// TIA Portal V19 export
// export: Created 2024-12-12T07:14:07.305667Z, ExportSetting WithDefaults, DisplayName Totally Integrated Automation Portal, DisplayVersion V19 Update 1, DisplayName TIA Portal Openness, DisplayVersion V19 Update 1, DisplayName TIA Portal Version Control Interface, DisplayVersion V19, DisplayName SINAMICS Startdrive Advanced, DisplayVersion V19, DisplayName SINAMICS DCC, DisplayVersion V19, DisplayName SINAMICS Startdrive G130, G150, S120, S150, SINAMICS MV, G220, S200, S210, DisplayVersion V19, DisplayName SINAMICS Startdrive G110M, G120, G120C, G120D, G120P, G115D, DisplayVersion V19, DisplayName STEP 7 Professional, DisplayVersion V19 Update 1, DisplayName STEP 7 Safety, DisplayVersion V19 Update 1, DisplayName WinCC Advanced, DisplayVersion V19 Update 1, DisplayName WinCC Advanced / Unified PC, DisplayVersion V19 Update 1
DATA_BLOCK "CW1"   // DB218
{ S7_Optimized_Access := 'TRUE' }
VERSION : 0.1
// stored: AutoNumber true, DBAccessibleFromOPCUA true, DBAccessibleFromWebserver true, InstanceOfName EM_CWM, InstanceOfType UDT, IsOnlyStoredInLoadMemory false, IsWriteProtectedInAS false
"EM_CWM"
   // VAR RETAIN
   //    Std : "EM_Std";
   //    Param : "EM_CWM_Param";
   //    LastHmiDataParam : "EM_CWM_Param";
   //    Alm : "EM_CWM_Alm";
   //    AlmWinCC : "EM_CWM_AlmWinCC";
   //    Sign : "EM_Sign";
   //    SignWinCC : "EM_Sign_WinCC";
   //    Input : "EM_CWM_Input";
   //    Output : "EM_CWM_Output";
   //    ExchangeFromChain : "EM_CWM_Exchange_FromChain";
   //    ExchangeToChain : "EM_CWM_Exchange_ToChain";
   //    Scale : "Scale_Wipotec";
   // END_VAR
BEGIN
   Std.Cfg_ModuleSync := TRUE;
   Std.Cfg_0_BelongShort_1_BelongLong := TRUE;
   Std.Cfg_ExternalCPU := FALSE;
   Std.Cfg_0_JogWord_1_JogBit := TRUE;
   Std._0_PriorityAlm_1_FirstAlm := FALSE;
   Std.AbortAlmOk := TRUE;
   Std.ServicesAbortAlmOk := TRUE;
   Std.SignOK := TRUE;
   Std.AlmReset := FALSE;
   Std.SignReset := FALSE;
   Std.NewAlm := FALSE;
   Std.NewSign := FALSE;
   Std.RstNewAlm := FALSE;
   Std.RstNewSign := FALSE;
   Std.AllowCopyByCategory := TRUE;
   Std.ForceCopyAll := FALSE;
   Std.InitCategories := FALSE;
   Std.InitCauses := FALSE;
   Std.Diag_AlmFound := FALSE;
   Std.Diag_SignFound := FALSE;
   Std.ScOk := TRUE;
   Std.OkToStop := TRUE;
   Std.PwrDrv := TRUE;
   Std.DriveRunCmd := FALSE;
   Std.ManAct := FALSE;
   Std.MachineSelected := TRUE;
   Std.MachineExtracted := FALSE;
   Std.LocalAbortReq := FALSE;
   Std.CondOkToEnaStaReq := FALSE;
   Std.EnaReq := FALSE;
   Std.EnaStaReq := FALSE;
   Std.StaReq := FALSE;
   Std.ReqStart := FALSE;
   Std.ReqStop := FALSE;
   Std.ReqAbort := TRUE;
   Std.ReqExecute := FALSE;
   Std.ReqReset := FALSE;
   Std.ReqSuspend := FALSE;
   Std.ReqUnSuspend := FALSE;
   Std.StrobeDeviceDiag := TRUE;
   Std.StrobeInverterDiag := FALSE;
   Std.DeviceDiagnosticDone := FALSE;
   Std.InverterDiagnosticDone := FALSE;
   Std.RecipeOnlineLoadDone := FALSE;
   Std.RecipeOnlineSaveDone := FALSE;
   Std.RecipeOfflineLoadDone := FALSE;
   Std.RecipeOfflineSaveDone := FALSE;
   Std.LastHmiDataLoadDone := FALSE;
   Std.LastHmiDataSaveDone := FALSE;
   Std.SummAlmTimeoutStart := FALSE;
   Std.SirenEna := FALSE;
   Std.VisEnButtons := TRUE;
   Std.VisManButtons := FALSE;
   Std.VisHomeButtons := FALSE;
   Std.VisEnButtonsRunning := TRUE;
   Std.Ena_Suspended := TRUE;
   Std.BluStkLgh_Steady_Cond := FALSE;
   Std.BluStkLgh_Frequency1_Cond := FALSE;
   Std.Siren_Frequency4_Cond := FALSE;
   Std.Cfg_ModuleNumber := 5;
   Std.Cfg_DeviceDiagCounter_Preset := 1;
   Std.Cfg_InverterDiagCounter_Preset := 0;
   Std.Cfg_Num_AlmDint := 8;
   Std.Cfg_Num_SignDint := 3;
   Std.Cfg_StaPbt := 65535;
   Std.Cfg_StoPbt := 65535;
   Std.Cfg_RstPbt := -1;
   Std.Cfg_EnaPbt := 65535;
   Std.Cfg_Siren := 1;
   Std.Cfg_Stack := 1;
   Std.Cfg_DisableStates[0..31] := 0;
   Std.Cfg_ModeTransitions[0..31] := 0;
   Std.Cfg_ModeNames[0..31] := '';
   Std.ModeCurrentName := 'Production';
   Std.StateCurrentName := 'Aborted';
   Std.DeviceDiagCounter := 1;
   Std.InverterDiagCounter := 0;
   Std.MaintenanceActivated."0" := FALSE;
   Std.MaintenanceActivated."1" := FALSE;
   Std.MaintenanceActivated."2" := FALSE;
   Std.MaintenanceActivated."3" := FALSE;
   Std.MaintenanceActivated."4" := FALSE;
   Std.MaintenanceActivated."5" := FALSE;
   Std.MaintenanceActivated."6" := FALSE;
   Std.MaintenanceActivated."7" := FALSE;
   Std.MaintenanceActivated."8" := FALSE;
   Std.MaintenanceActivated."9" := FALSE;
   Std.MaintenanceActivated."10" := FALSE;
   Std.MaintenanceActivated."11" := FALSE;
   Std.MaintenanceActivated."12" := FALSE;
   Std.MaintenanceActivated."13" := FALSE;
   Std.MaintenanceActivated."14" := FALSE;
   Std.MaintenanceActivated."15" := FALSE;
   Std.MaintenanceActivated."16" := FALSE;
   Std.MaintenanceActivated."17" := FALSE;
   Std.MaintenanceActivated."18" := FALSE;
   Std.MaintenanceActivated."19" := FALSE;
   Std.MaintenanceActivated."20" := FALSE;
   Std.MaintenanceActivated."21" := FALSE;
   Std.MaintenanceActivated."22" := FALSE;
   Std.MaintenanceActivated."23" := FALSE;
   Std.MaintenanceActivated."24" := FALSE;
   Std.MaintenanceActivated."25" := FALSE;
   Std.MaintenanceActivated."26" := FALSE;
   Std.MaintenanceActivated."27" := FALSE;
   Std.MaintenanceActivated."28" := FALSE;
   Std.MaintenanceActivated."29" := FALSE;
   Std.MaintenanceActivated."30" := FALSE;
   Std.MaintenanceActivated."31" := FALSE;
   Std.MaintenanceReq."0" := FALSE;
   Std.MaintenanceReq."1" := FALSE;
   Std.MaintenanceReq."2" := FALSE;
   Std.MaintenanceReq."3" := FALSE;
   Std.MaintenanceReq."4" := FALSE;
   Std.MaintenanceReq."5" := FALSE;
   Std.MaintenanceReq."6" := FALSE;
   Std.MaintenanceReq."7" := FALSE;
   Std.MaintenanceReq."8" := FALSE;
   Std.MaintenanceReq."9" := FALSE;
   Std.MaintenanceReq."10" := FALSE;
   Std.MaintenanceReq."11" := FALSE;
   Std.MaintenanceReq."12" := FALSE;
   Std.MaintenanceReq."13" := FALSE;
   Std.MaintenanceReq."14" := FALSE;
   Std.MaintenanceReq."15" := FALSE;
   Std.MaintenanceReq."16" := FALSE;
   Std.MaintenanceReq."17" := FALSE;
   Std.MaintenanceReq."18" := FALSE;
   Std.MaintenanceReq."19" := FALSE;
   Std.MaintenanceReq."20" := FALSE;
   Std.MaintenanceReq."21" := FALSE;
   Std.MaintenanceReq."22" := FALSE;
   Std.MaintenanceReq."23" := FALSE;
   Std.MaintenanceReq."24" := FALSE;
   Std.MaintenanceReq."25" := FALSE;
   Std.MaintenanceReq."26" := FALSE;
   Std.MaintenanceReq."27" := FALSE;
   Std.MaintenanceReq."28" := FALSE;
   Std.MaintenanceReq."29" := FALSE;
   Std.MaintenanceReq."30" := FALSE;
   Std.MaintenanceReq."31" := FALSE;
   Std.WithinScreenRange := 0;
   Std.ExchangeToGlobal.Communication.RunMode := FALSE;
   Std.ExchangeToGlobal.Communication.ConnectionFaulted := FALSE;
   Std.ExchangeToGlobal.Gen.Communication := FALSE;
   Std.ExchangeToGlobal.Gen.Selected := TRUE;
   Std.ExchangeToGlobal.Gen.Extracted := FALSE;
   Std.ExchangeToGlobal.Gen.EnaReq := FALSE;
   Std.ExchangeToGlobal.Gen.StaReq := FALSE;
   Std.ExchangeToGlobal.Gen.Started := FALSE;
   Std.ExchangeToGlobal.Gen.Unsuspended := FALSE;
   Std.ExchangeToGlobal.Gen.Ena_Suspended := TRUE;
   Std.ExchangeToGlobal.Gen.sts_Starting := FALSE;
   Std.ExchangeToGlobal.Gen.sts_Stopping := FALSE;
   Std.ExchangeToGlobal.Gen.sts_Aborting := FALSE;
   Std.ExchangeToGlobal.Gen.sts_Suspending := FALSE;
   Std.ExchangeToGlobal.Gen.sts_Unsuspending := FALSE;
   Std.ExchangeToGlobal.Gen.sts_Execute := FALSE;
   Std.ExchangeToGlobal.Gen.sts_Idle := FALSE;
   Std.ExchangeToGlobal.Gen.sts_Stopped := FALSE;
   Std.ExchangeToGlobal.Gen.sts_Aborted := TRUE;
   Std.ExchangeToGlobal.Gen.sts_Suspended := FALSE;
   Std.ExchangeToGlobal.Gen.sts_ModeManual := FALSE;
   Std.ExchangeToGlobal.Gen.sts_ModeAutomatic := TRUE;
   Std.ExchangeToGlobal.Gen.NewAlm := FALSE;
   Std.ExchangeToGlobal.Gen.NewSign := FALSE;
   Std.ExchangeToGlobal.Gen.RecipeOnlineLoadDone := FALSE;
   Std.ExchangeToGlobal.Gen.RecipeOnlineSaveDone := FALSE;
   Std.ExchangeToGlobal.Gen.RecipeOfflineLoadDone := FALSE;
   Std.ExchangeToGlobal.Gen.RecipeOfflineSaveDone := FALSE;
   Std.ExchangeToGlobal.Gen.LastHmiDataLoadDone := FALSE;
   Std.ExchangeToGlobal.Gen.LastHmiDataSaveDone := FALSE;
   Std.ExchangeToGlobal.Gen.InverterDiagnosticDone := FALSE;
   Std.ExchangeToGlobal.Gen.AxisGroupSync := TRUE;
   Std.ExchangeToGlobal.Gen.CmdMode := 1;
   Std.ExchangeToGlobal.Gen.Mode := 1;
   Std.ExchangeToGlobal.Gen.DisableEnaPbt := 0;
   Std.ExchangeToGlobal.Input.StaPbt := FALSE;
   Std.ExchangeToGlobal.Input.StoPbt := FALSE;
   Std.ExchangeToGlobal.Input.RstPbt := FALSE;
   Std.ExchangeToGlobal.Input.EnaPbt := FALSE;
   Std.ExchangeToGlobal.Input._4 := FALSE;
   Std.ExchangeToGlobal.Input._5 := FALSE;
   Std.ExchangeToGlobal.Input._6 := FALSE;
   Std.ExchangeToGlobal.Input._7 := FALSE;
   Std.ExchangeToGlobal.Input._8 := FALSE;
   Std.ExchangeToGlobal.Input._9 := FALSE;
   Std.ExchangeToGlobal.Input._10 := FALSE;
   Std.ExchangeToGlobal.Input._11 := FALSE;
   Std.ExchangeToGlobal.Input._12 := FALSE;
   Std.ExchangeToGlobal.Input._13 := FALSE;
   Std.ExchangeToGlobal.Input._14 := FALSE;
   Std.ExchangeToGlobal.Input._15 := FALSE;
   Std.ExchangeToGlobal.AlmOk.ThSwitch := TRUE;
   Std.ExchangeToGlobal.AlmOk.SafeComm := TRUE;
   Std.ExchangeToGlobal.AlmOk.SafeEmg := TRUE;
   Std.ExchangeToGlobal.AlmOk.SafeGuards := TRUE;
   Std.ExchangeToGlobal.AlmOk.GtaAirGroup := TRUE;
   Std.ExchangeToGlobal.AlmOk.Major := TRUE;
   Std.ExchangeToGlobal.AlmOk.Minor := TRUE;
   Std.ExchangeToGlobal.AlmOk.Spare07 := TRUE;
   Std.ExchangeToGlobal.AlmOk.Spare08 := TRUE;
   Std.ExchangeToGlobal.AlmOk.Spare09 := TRUE;
   Std.ExchangeToGlobal.AlmOk.Spare10 := TRUE;
   Std.ExchangeToGlobal.AlmOk.Spare11 := TRUE;
   Std.ExchangeToGlobal.AlmOk.Spare12 := TRUE;
   Std.ExchangeToGlobal.AlmOk.Spare13 := TRUE;
   Std.ExchangeToGlobal.AlmOk.Spare14 := TRUE;
   Std.ExchangeToGlobal.AlmOk.Spare15 := TRUE;
   Std.ExchangeToGlobal.AlmOk.Spare16 := TRUE;
   Std.ExchangeToGlobal.AlmOk.Spare17 := TRUE;
   Std.ExchangeToGlobal.AlmOk.Spare18 := TRUE;
   Std.ExchangeToGlobal.AlmOk.Spare19 := TRUE;
   Std.ExchangeToGlobal.AlmOk.Spare20 := TRUE;
   Std.ExchangeToGlobal.AlmOk.Spare21 := TRUE;
   Std.ExchangeToGlobal.AlmOk.Spare22 := TRUE;
   Std.ExchangeToGlobal.AlmOk.Spare23 := TRUE;
   Std.ExchangeToGlobal.AlmOk.Spare24 := TRUE;
   Std.ExchangeToGlobal.AlmOk.Spare25 := TRUE;
   Std.ExchangeToGlobal.AlmOk.Spare26 := TRUE;
   Std.ExchangeToGlobal.AlmOk.Spare27 := TRUE;
   Std.ExchangeToGlobal.AlmOk.Spare28 := TRUE;
   Std.ExchangeToGlobal.AlmOk.Spare29 := TRUE;
   Std.ExchangeToGlobal.AlmOk.Spare30 := TRUE;
   Std.ExchangeToGlobal.AlmOk.Spare31 := TRUE;
   Std.ExchangeToGlobal.AlmCauseOk.Ope := TRUE;
   Std.ExchangeToGlobal.AlmCauseOk.Ust := TRUE;
   Std.ExchangeToGlobal.AlmCauseOk.Dst := TRUE;
   Std.ExchangeToGlobal.AlmCauseOk.Ext := TRUE;
   Std.ExchangeToGlobal.AlmCauseOk.Mac := TRUE;
   Std.ExchangeToGlobal.AlmCauseOk.Spare05 := TRUE;
   Std.ExchangeToGlobal.AlmCauseOk.Spare06 := TRUE;
   Std.ExchangeToGlobal.AlmCauseOk.Spare07 := TRUE;
   Std.ExchangeToGlobal.AlmCauseOk.Spare08 := TRUE;
   Std.ExchangeToGlobal.AlmCauseOk.Spare09 := TRUE;
   Std.ExchangeToGlobal.AlmCauseOk.Spare10 := TRUE;
   Std.ExchangeToGlobal.AlmCauseOk.Spare11 := TRUE;
   Std.ExchangeToGlobal.AlmCauseOk.Spare12 := TRUE;
   Std.ExchangeToGlobal.AlmCauseOk.Spare13 := TRUE;
   Std.ExchangeToGlobal.AlmCauseOk.Spare14 := TRUE;
   Std.ExchangeToGlobal.AlmCauseOk.Spare15 := TRUE;
   Std.ExchangeToGlobal.AlmCauseOk.Spare16 := TRUE;
   Std.ExchangeToGlobal.AlmCauseOk.Spare17 := TRUE;
   Std.ExchangeToGlobal.AlmCauseOk.Spare18 := TRUE;
   Std.ExchangeToGlobal.AlmCauseOk.Spare19 := TRUE;
   Std.ExchangeToGlobal.AlmCauseOk.Spare20 := TRUE;
   Std.ExchangeToGlobal.AlmCauseOk.Spare21 := TRUE;
   Std.ExchangeToGlobal.AlmCauseOk.Spare22 := TRUE;
   Std.ExchangeToGlobal.AlmCauseOk.Spare23 := TRUE;
   Std.ExchangeToGlobal.AlmCauseOk.Spare24 := TRUE;
   Std.ExchangeToGlobal.AlmCauseOk.Spare25 := TRUE;
   Std.ExchangeToGlobal.AlmCauseOk.Spare26 := TRUE;
   Std.ExchangeToGlobal.AlmCauseOk.Spare27 := TRUE;
   Std.ExchangeToGlobal.AlmCauseOk.Spare28 := TRUE;
   Std.ExchangeToGlobal.AlmCauseOk.Spare29 := TRUE;
   Std.ExchangeToGlobal.AlmCauseOk.Spare30 := TRUE;
   Std.ExchangeToGlobal.AlmCauseOk.Spare31 := TRUE;
   Std.ExchangeToGlobal.AlmBannerFbk.FirstAlmDetection := FALSE;
   Std.ExchangeToGlobal.AlmBannerFbk.AlmPriority := 100;
   Std.ExchangeToGlobal.AlmBannerFbk.AlmCategory := -1;
   Std.ExchangeToGlobal.AlmBannerFbk.AlmCause := -1;
   Std.ExchangeToGlobal.AlmBannerFbk.AlmID := -1;
   Std.ExchangeToGlobal.AlmBannerFbk.GlobalAbsTime := 0;
   Std.ExchangeToGlobal.SignBannerFbk.SignPriority := 100;
   Std.ExchangeToGlobal.SignBannerFbk.SignCategory := -1;
   Std.ExchangeToGlobal.SignBannerFbk.SignID := -1;
   Std.ExchangeToGlobal.ExtCPU.PushButton.StaPbt := FALSE;
   Std.ExchangeToGlobal.ExtCPU.PushButton.StoPbt := FALSE;
   Std.ExchangeToGlobal.ExtCPU.PushButton.RstPbt := FALSE;
   Std.ExchangeToGlobal.ExtCPU.PushButton.EnaPbt := FALSE;
   Std.ExchangeToGlobal.ExtCPU.PushButton.EnaReq := FALSE;
   Std.ExchangeToGlobal.ExtCPU.PushButton.EnaStaReq := FALSE;
   Std.ExchangeToGlobal.ExtCPU.DeviceDiagDone := FALSE;
   Std.ExchangeToGlobal.ExtCPU.InverterDiagDone := FALSE;
   Std.ExchangeToGlobal.LightSiren.Cfg_StaPbt := 65535;
   Std.ExchangeToGlobal.LightSiren.Cfg_RstPbt := -1;
   Std.ExchangeToGlobal.LightSiren.Cfg_EnaPbt := 65535;
   Std.ExchangeToGlobal.LightSiren.Cfg_Siren := 1;
   Std.ExchangeToGlobal.LightSiren.Cfg_Stack := 1;
   Std.ExchangeToGlobal.LightSiren.Steady.StaPbtLgh := FALSE;
   Std.ExchangeToGlobal.LightSiren.Steady.RstPbtLgh := FALSE;
   Std.ExchangeToGlobal.LightSiren.Steady.EnaPbtLgh := FALSE;
   Std.ExchangeToGlobal.LightSiren.Steady.Siren := FALSE;
   Std.ExchangeToGlobal.LightSiren.Steady.YelStkLgh := FALSE;
   Std.ExchangeToGlobal.LightSiren.Steady.BluStkLgh := FALSE;
   Std.ExchangeToGlobal.LightSiren.Steady.GrnStkLgh := FALSE;
   Std.ExchangeToGlobal.LightSiren.Steady.WhtStkLgh := FALSE;
   Std.ExchangeToGlobal.LightSiren.Steady.Cust1_StaPbtLgh := FALSE;
   Std.ExchangeToGlobal.LightSiren.Steady.Cust1_RstPbtLgh := FALSE;
   Std.ExchangeToGlobal.LightSiren.Steady.Cust1_Siren := FALSE;
   Std.ExchangeToGlobal.LightSiren.Steady.Cust1_RedStkLgh := FALSE;
   Std.ExchangeToGlobal.LightSiren.Steady.Cust1_OngStkLgh := FALSE;
   Std.ExchangeToGlobal.LightSiren.Steady.Cust1_GrnStkLgh := FALSE;
   Std.ExchangeToGlobal.LightSiren.Steady.Cust1_BluStkLgh := FALSE;
   Std.ExchangeToGlobal.LightSiren.Steady.Cust1_WhtStkLgh := FALSE;
   Std.ExchangeToGlobal.LightSiren.Frequency1.StaPbtLgh := FALSE;
   Std.ExchangeToGlobal.LightSiren.Frequency1.RstPbtLgh := FALSE;
   Std.ExchangeToGlobal.LightSiren.Frequency1.EnaPbtLgh := FALSE;
   Std.ExchangeToGlobal.LightSiren.Frequency1.Siren := FALSE;
   Std.ExchangeToGlobal.LightSiren.Frequency1.YelStkLgh := FALSE;
   Std.ExchangeToGlobal.LightSiren.Frequency1.BluStkLgh := FALSE;
   Std.ExchangeToGlobal.LightSiren.Frequency1.GrnStkLgh := FALSE;
   Std.ExchangeToGlobal.LightSiren.Frequency1.WhtStkLgh := FALSE;
   Std.ExchangeToGlobal.LightSiren.Frequency1.Cust1_StaPbtLgh := FALSE;
   Std.ExchangeToGlobal.LightSiren.Frequency1.Cust1_RstPbtLgh := FALSE;
   Std.ExchangeToGlobal.LightSiren.Frequency1.Cust1_Siren := FALSE;
   Std.ExchangeToGlobal.LightSiren.Frequency1.Cust1_RedStkLgh := FALSE;
   Std.ExchangeToGlobal.LightSiren.Frequency1.Cust1_OngStkLgh := FALSE;
   Std.ExchangeToGlobal.LightSiren.Frequency1.Cust1_GrnStkLgh := FALSE;
   Std.ExchangeToGlobal.LightSiren.Frequency1.Cust1_BluStkLgh := FALSE;
   Std.ExchangeToGlobal.LightSiren.Frequency1.Cust1_WhtStkLgh := FALSE;
   Std.ExchangeToGlobal.LightSiren.Frequency2.StaPbtLgh := FALSE;
   Std.ExchangeToGlobal.LightSiren.Frequency2.RstPbtLgh := FALSE;
   Std.ExchangeToGlobal.LightSiren.Frequency2.EnaPbtLgh := FALSE;
   Std.ExchangeToGlobal.LightSiren.Frequency2.Siren := FALSE;
   Std.ExchangeToGlobal.LightSiren.Frequency2.YelStkLgh := FALSE;
   Std.ExchangeToGlobal.LightSiren.Frequency2.BluStkLgh := FALSE;
   Std.ExchangeToGlobal.LightSiren.Frequency2.GrnStkLgh := FALSE;
   Std.ExchangeToGlobal.LightSiren.Frequency2.WhtStkLgh := FALSE;
   Std.ExchangeToGlobal.LightSiren.Frequency2.Cust1_StaPbtLgh := FALSE;
   Std.ExchangeToGlobal.LightSiren.Frequency2.Cust1_RstPbtLgh := FALSE;
   Std.ExchangeToGlobal.LightSiren.Frequency2.Cust1_Siren := FALSE;
   Std.ExchangeToGlobal.LightSiren.Frequency2.Cust1_RedStkLgh := FALSE;
   Std.ExchangeToGlobal.LightSiren.Frequency2.Cust1_OngStkLgh := FALSE;
   Std.ExchangeToGlobal.LightSiren.Frequency2.Cust1_GrnStkLgh := FALSE;
   Std.ExchangeToGlobal.LightSiren.Frequency2.Cust1_BluStkLgh := FALSE;
   Std.ExchangeToGlobal.LightSiren.Frequency2.Cust1_WhtStkLgh := FALSE;
   Std.ExchangeToGlobal.LightSiren.Frequency3.StaPbtLgh := FALSE;
   Std.ExchangeToGlobal.LightSiren.Frequency3.RstPbtLgh := FALSE;
   Std.ExchangeToGlobal.LightSiren.Frequency3.EnaPbtLgh := FALSE;
   Std.ExchangeToGlobal.LightSiren.Frequency3.Siren := FALSE;
   Std.ExchangeToGlobal.LightSiren.Frequency3.YelStkLgh := FALSE;
   Std.ExchangeToGlobal.LightSiren.Frequency3.BluStkLgh := FALSE;
   Std.ExchangeToGlobal.LightSiren.Frequency3.GrnStkLgh := FALSE;
   Std.ExchangeToGlobal.LightSiren.Frequency3.WhtStkLgh := FALSE;
   Std.ExchangeToGlobal.LightSiren.Frequency3.Cust1_StaPbtLgh := FALSE;
   Std.ExchangeToGlobal.LightSiren.Frequency3.Cust1_RstPbtLgh := FALSE;
   Std.ExchangeToGlobal.LightSiren.Frequency3.Cust1_Siren := FALSE;
   Std.ExchangeToGlobal.LightSiren.Frequency3.Cust1_RedStkLgh := FALSE;
   Std.ExchangeToGlobal.LightSiren.Frequency3.Cust1_OngStkLgh := FALSE;
   Std.ExchangeToGlobal.LightSiren.Frequency3.Cust1_GrnStkLgh := FALSE;
   Std.ExchangeToGlobal.LightSiren.Frequency3.Cust1_BluStkLgh := FALSE;
   Std.ExchangeToGlobal.LightSiren.Frequency3.Cust1_WhtStkLgh := FALSE;
   Std.ExchangeToGlobal.LightSiren.Frequency4.StaPbtLgh := FALSE;
   Std.ExchangeToGlobal.LightSiren.Frequency4.RstPbtLgh := FALSE;
   Std.ExchangeToGlobal.LightSiren.Frequency4.EnaPbtLgh := FALSE;
   Std.ExchangeToGlobal.LightSiren.Frequency4.Siren := FALSE;
   Std.ExchangeToGlobal.LightSiren.Frequency4.YelStkLgh := FALSE;
   Std.ExchangeToGlobal.LightSiren.Frequency4.BluStkLgh := FALSE;
   Std.ExchangeToGlobal.LightSiren.Frequency4.GrnStkLgh := FALSE;
   Std.ExchangeToGlobal.LightSiren.Frequency4.WhtStkLgh := FALSE;
   Std.ExchangeToGlobal.LightSiren.Frequency4.Cust1_StaPbtLgh := FALSE;
   Std.ExchangeToGlobal.LightSiren.Frequency4.Cust1_RstPbtLgh := FALSE;
   Std.ExchangeToGlobal.LightSiren.Frequency4.Cust1_Siren := FALSE;
   Std.ExchangeToGlobal.LightSiren.Frequency4.Cust1_RedStkLgh := FALSE;
   Std.ExchangeToGlobal.LightSiren.Frequency4.Cust1_OngStkLgh := FALSE;
   Std.ExchangeToGlobal.LightSiren.Frequency4.Cust1_GrnStkLgh := FALSE;
   Std.ExchangeToGlobal.LightSiren.Frequency4.Cust1_BluStkLgh := FALSE;
   Std.ExchangeToGlobal.LightSiren.Frequency4.Cust1_WhtStkLgh := FALSE;
   Std.ExchangeToGlobal.PackML.Sts_Aborted := TRUE;
   Std.ExchangeToGlobal.PackML.Sts_Aborting := FALSE;
   Std.ExchangeToGlobal.PackML.Sts_Clearing := FALSE;
   Std.ExchangeToGlobal.PackML.Sts_Complete := FALSE;
   Std.ExchangeToGlobal.PackML.Sts_Completing := FALSE;
   Std.ExchangeToGlobal.PackML.Sts_Execute := FALSE;
   Std.ExchangeToGlobal.PackML.Sts_Held := FALSE;
   Std.ExchangeToGlobal.PackML.Sts_Holding := FALSE;
   Std.ExchangeToGlobal.PackML.Sts_Idle := FALSE;
   Std.ExchangeToGlobal.PackML.Sts_Resetting := FALSE;
   Std.ExchangeToGlobal.PackML.Sts_Starting := FALSE;
   Std.ExchangeToGlobal.PackML.Sts_Stopped := FALSE;
   Std.ExchangeToGlobal.PackML.Sts_Stopping := FALSE;
   Std.ExchangeToGlobal.PackML.Sts_Suspended := FALSE;
   Std.ExchangeToGlobal.PackML.Sts_Suspending := FALSE;
   Std.ExchangeToGlobal.PackML.Sts_UnHolding := FALSE;
   Std.ExchangeToGlobal.PackML.Sts_UnSuspending := FALSE;
   Std.ExchangeToGlobal.PackML.Sts_AbortedEnabled := TRUE;
   Std.ExchangeToGlobal.PackML.Sts_AbortingEnabled := TRUE;
   Std.ExchangeToGlobal.PackML.Sts_ClearingEnabled := TRUE;
   Std.ExchangeToGlobal.PackML.Sts_CompleteEnabled := FALSE;
   Std.ExchangeToGlobal.PackML.Sts_CompletingEnabled := FALSE;
   Std.ExchangeToGlobal.PackML.Sts_ExecuteEnabled := TRUE;
   Std.ExchangeToGlobal.PackML.Sts_HeldEnabled := FALSE;
   Std.ExchangeToGlobal.PackML.Sts_HoldingEnabled := FALSE;
   Std.ExchangeToGlobal.PackML.Sts_IdleEnabled := TRUE;
   Std.ExchangeToGlobal.PackML.Sts_ResettingEnabled := TRUE;
   Std.ExchangeToGlobal.PackML.Sts_StartingEnabled := TRUE;
   Std.ExchangeToGlobal.PackML.Sts_StoppedEnabled := TRUE;
   Std.ExchangeToGlobal.PackML.Sts_StoppingEnabled := TRUE;
   Std.ExchangeToGlobal.PackML.Sts_SuspendedEnabled := TRUE;
   Std.ExchangeToGlobal.PackML.Sts_SuspendingEnabled := TRUE;
   Std.ExchangeToGlobal.PackML.Sts_UnHoldingEnabled := FALSE;
   Std.ExchangeToGlobal.PackML.Sts_UnSuspendingEnabled := TRUE;
   Std.ExchangeToGlobal.SignOk := TRUE;
   Std.ExchangeToGlobal."Dint"[0..4] := 0;
   Std.VisAlmTypeBool.ThSwitch := FALSE;
   Std.VisAlmTypeBool.SafeComm := FALSE;
   Std.VisAlmTypeBool.SafeEmg := FALSE;
   Std.VisAlmTypeBool.SafeGuards := TRUE;
   Std.VisAlmTypeBool.GtaAirGroup := FALSE;
   Std.VisAlmTypeBool.Major := FALSE;
   Std.VisAlmTypeBool.Minor := FALSE;
   Std.VisAlmTypeBool.Spare07 := FALSE;
   Std.VisAlmTypeBool.Spare08 := FALSE;
   Std.VisAlmTypeBool.Spare09 := FALSE;
   Std.VisAlmTypeBool.Spare10 := FALSE;
   Std.VisAlmTypeBool.Spare11 := FALSE;
   Std.VisAlmTypeBool.Spare12 := FALSE;
   Std.VisAlmTypeBool.Spare13 := FALSE;
   Std.VisAlmTypeBool.Spare14 := FALSE;
   Std.VisAlmTypeBool.Spare15 := FALSE;
   Std.VisAlmTypeBool.Spare16 := FALSE;
   Std.VisAlmTypeBool.Spare17 := FALSE;
   Std.VisAlmTypeBool.Spare18 := FALSE;
   Std.VisAlmTypeBool.Spare19 := FALSE;
   Std.VisAlmTypeBool.Spare20 := FALSE;
   Std.VisAlmTypeBool.Spare21 := FALSE;
   Std.VisAlmTypeBool.Spare22 := FALSE;
   Std.VisAlmTypeBool.Spare23 := FALSE;
   Std.VisAlmTypeBool.Spare24 := FALSE;
   Std.VisAlmTypeBool.Spare25 := FALSE;
   Std.VisAlmTypeBool.Spare26 := FALSE;
   Std.VisAlmTypeBool.Spare27 := FALSE;
   Std.VisAlmTypeBool.Spare28 := FALSE;
   Std.VisAlmTypeBool.Spare29 := FALSE;
   Std.VisAlmTypeBool.Spare30 := FALSE;
   Std.VisAlmTypeBool.Spare31 := FALSE;
   Std.AlmTypeFbk.ThSwitch := FALSE;
   Std.AlmTypeFbk.SafeComm := FALSE;
   Std.AlmTypeFbk.SafeEmg := FALSE;
   Std.AlmTypeFbk.SafeGuards := FALSE;
   Std.AlmTypeFbk.GtaAirGroup := FALSE;
   Std.AlmTypeFbk.Major := FALSE;
   Std.AlmTypeFbk.Minor := FALSE;
   Std.AlmTypeFbk.Spare07 := FALSE;
   Std.AlmTypeFbk.Spare08 := FALSE;
   Std.AlmTypeFbk.Spare09 := FALSE;
   Std.AlmTypeFbk.Spare10 := FALSE;
   Std.AlmTypeFbk.Spare11 := FALSE;
   Std.AlmTypeFbk.Spare12 := FALSE;
   Std.AlmTypeFbk.Spare13 := FALSE;
   Std.AlmTypeFbk.Spare14 := FALSE;
   Std.AlmTypeFbk.Spare15 := FALSE;
   Std.AlmTypeFbk.Spare16 := FALSE;
   Std.AlmTypeFbk.Spare17 := FALSE;
   Std.AlmTypeFbk.Spare18 := FALSE;
   Std.AlmTypeFbk.Spare19 := FALSE;
   Std.AlmTypeFbk.Spare20 := FALSE;
   Std.AlmTypeFbk.Spare21 := FALSE;
   Std.AlmTypeFbk.Spare22 := FALSE;
   Std.AlmTypeFbk.Spare23 := FALSE;
   Std.AlmTypeFbk.Spare24 := FALSE;
   Std.AlmTypeFbk.Spare25 := FALSE;
   Std.AlmTypeFbk.Spare26 := FALSE;
   Std.AlmTypeFbk.Spare27 := FALSE;
   Std.AlmTypeFbk.Spare28 := FALSE;
   Std.AlmTypeFbk.Spare29 := FALSE;
   Std.AlmTypeFbk.Spare30 := FALSE;
   Std.AlmTypeFbk.Spare31 := FALSE;
   Std.AlmTypeOk.ThSwitch := TRUE;
   Std.AlmTypeOk.SafeComm := TRUE;
   Std.AlmTypeOk.SafeEmg := TRUE;
   Std.AlmTypeOk.SafeGuards := TRUE;
   Std.AlmTypeOk.GtaAirGroup := TRUE;
   Std.AlmTypeOk.Major := TRUE;
   Std.AlmTypeOk.Minor := TRUE;
   Std.AlmTypeOk.Spare07 := TRUE;
   Std.AlmTypeOk.Spare08 := TRUE;
   Std.AlmTypeOk.Spare09 := TRUE;
   Std.AlmTypeOk.Spare10 := TRUE;
   Std.AlmTypeOk.Spare11 := TRUE;
   Std.AlmTypeOk.Spare12 := TRUE;
   Std.AlmTypeOk.Spare13 := TRUE;
   Std.AlmTypeOk.Spare14 := TRUE;
   Std.AlmTypeOk.Spare15 := TRUE;
   Std.AlmTypeOk.Spare16 := TRUE;
   Std.AlmTypeOk.Spare17 := TRUE;
   Std.AlmTypeOk.Spare18 := TRUE;
   Std.AlmTypeOk.Spare19 := TRUE;
   Std.AlmTypeOk.Spare20 := TRUE;
   Std.AlmTypeOk.Spare21 := TRUE;
   Std.AlmTypeOk.Spare22 := TRUE;
   Std.AlmTypeOk.Spare23 := TRUE;
   Std.AlmTypeOk.Spare24 := TRUE;
   Std.AlmTypeOk.Spare25 := TRUE;
   Std.AlmTypeOk.Spare26 := TRUE;
   Std.AlmTypeOk.Spare27 := TRUE;
   Std.AlmTypeOk.Spare28 := TRUE;
   Std.AlmTypeOk.Spare29 := TRUE;
   Std.AlmTypeOk.Spare30 := TRUE;
   Std.AlmTypeOk.Spare31 := TRUE;
   Std.AlmCauseFbk.Ope := FALSE;
   Std.AlmCauseFbk.Ust := FALSE;
   Std.AlmCauseFbk.Dst := FALSE;
   Std.AlmCauseFbk.Ext := FALSE;
   Std.AlmCauseFbk.Mac := FALSE;
   Std.AlmCauseFbk.Spare05 := FALSE;
   Std.AlmCauseFbk.Spare06 := FALSE;
   Std.AlmCauseFbk.Spare07 := FALSE;
   Std.AlmCauseFbk.Spare08 := FALSE;
   Std.AlmCauseFbk.Spare09 := FALSE;
   Std.AlmCauseFbk.Spare10 := FALSE;
   Std.AlmCauseFbk.Spare11 := FALSE;
   Std.AlmCauseFbk.Spare12 := FALSE;
   Std.AlmCauseFbk.Spare13 := FALSE;
   Std.AlmCauseFbk.Spare14 := FALSE;
   Std.AlmCauseFbk.Spare15 := FALSE;
   Std.AlmCauseFbk.Spare16 := FALSE;
   Std.AlmCauseFbk.Spare17 := FALSE;
   Std.AlmCauseFbk.Spare18 := FALSE;
   Std.AlmCauseFbk.Spare19 := FALSE;
   Std.AlmCauseFbk.Spare20 := FALSE;
   Std.AlmCauseFbk.Spare21 := FALSE;
   Std.AlmCauseFbk.Spare22 := FALSE;
   Std.AlmCauseFbk.Spare23 := FALSE;
   Std.AlmCauseFbk.Spare24 := FALSE;
   Std.AlmCauseFbk.Spare25 := FALSE;
   Std.AlmCauseFbk.Spare26 := FALSE;
   Std.AlmCauseFbk.Spare27 := FALSE;
   Std.AlmCauseFbk.Spare28 := FALSE;
   Std.AlmCauseFbk.Spare29 := FALSE;
   Std.AlmCauseFbk.Spare30 := FALSE;
   Std.AlmCauseFbk.Spare31 := FALSE;
   Std.AlmCauseOk.Ope := TRUE;
   Std.AlmCauseOk.Ust := TRUE;
   Std.AlmCauseOk.Dst := TRUE;
   Std.AlmCauseOk.Ext := TRUE;
   Std.AlmCauseOk.Mac := TRUE;
   Std.AlmCauseOk.Spare05 := TRUE;
   Std.AlmCauseOk.Spare06 := TRUE;
   Std.AlmCauseOk.Spare07 := TRUE;
   Std.AlmCauseOk.Spare08 := TRUE;
   Std.AlmCauseOk.Spare09 := TRUE;
   Std.AlmCauseOk.Spare10 := TRUE;
   Std.AlmCauseOk.Spare11 := TRUE;
   Std.AlmCauseOk.Spare12 := TRUE;
   Std.AlmCauseOk.Spare13 := TRUE;
   Std.AlmCauseOk.Spare14 := TRUE;
   Std.AlmCauseOk.Spare15 := TRUE;
   Std.AlmCauseOk.Spare16 := TRUE;
   Std.AlmCauseOk.Spare17 := TRUE;
   Std.AlmCauseOk.Spare18 := TRUE;
   Std.AlmCauseOk.Spare19 := TRUE;
   Std.AlmCauseOk.Spare20 := TRUE;
   Std.AlmCauseOk.Spare21 := TRUE;
   Std.AlmCauseOk.Spare22 := TRUE;
   Std.AlmCauseOk.Spare23 := TRUE;
   Std.AlmCauseOk.Spare24 := TRUE;
   Std.AlmCauseOk.Spare25 := TRUE;
   Std.AlmCauseOk.Spare26 := TRUE;
   Std.AlmCauseOk.Spare27 := TRUE;
   Std.AlmCauseOk.Spare28 := TRUE;
   Std.AlmCauseOk.Spare29 := TRUE;
   Std.AlmCauseOk.Spare30 := TRUE;
   Std.AlmCauseOk.Spare31 := TRUE;
   Std.ForceCategory.ThSwitch := FALSE;
   Std.ForceCategory.SafeComm := TRUE;
   Std.ForceCategory.SafeEmg := TRUE;
   Std.ForceCategory.SafeGuards := FALSE;
   Std.ForceCategory.GtaAirGroup := FALSE;
   Std.ForceCategory.Major := FALSE;
   Std.ForceCategory.Minor := FALSE;
   Std.ForceCategory.Spare07 := FALSE;
   Std.ForceCategory.Spare08 := FALSE;
   Std.ForceCategory.Spare09 := FALSE;
   Std.ForceCategory.Spare10 := FALSE;
   Std.ForceCategory.Spare11 := FALSE;
   Std.ForceCategory.Spare12 := FALSE;
   Std.ForceCategory.Spare13 := FALSE;
   Std.ForceCategory.Spare14 := FALSE;
   Std.ForceCategory.Spare15 := FALSE;
   Std.ForceCategory.Spare16 := FALSE;
   Std.ForceCategory.Spare17 := FALSE;
   Std.ForceCategory.Spare18 := FALSE;
   Std.ForceCategory.Spare19 := FALSE;
   Std.ForceCategory.Spare20 := FALSE;
   Std.ForceCategory.Spare21 := FALSE;
   Std.ForceCategory.Spare22 := FALSE;
   Std.ForceCategory.Spare23 := FALSE;
   Std.ForceCategory.Spare24 := FALSE;
   Std.ForceCategory.Spare25 := FALSE;
   Std.ForceCategory.Spare26 := FALSE;
   Std.ForceCategory.Spare27 := FALSE;
   Std.ForceCategory.Spare28 := FALSE;
   Std.ForceCategory.Spare29 := FALSE;
   Std.ForceCategory.Spare30 := FALSE;
   Std.ForceCategory.Spare31 := FALSE;
   Std.AlmStruct.Alm[0..31] := 0;
   Std.AlmStruct.Category[0..31] := 0;
   Std.AlmStruct.Category[32..63] := 1;
   Std.AlmStruct.Category[64..95] := 2;
   Std.AlmStruct.Category[96..127] := 3;
   Std.AlmStruct.Category[128..159] := 4;
   Std.AlmStruct.Category[160..191] := 5;
   Std.AlmStruct.Category[192..1023] := 6;
   Std.AlmStruct.BannerPriority[0..31] := 0;
   Std.AlmStruct.BannerPriority[32..63] := 1;
   Std.AlmStruct.BannerPriority[64..95] := 2;
   Std.AlmStruct.BannerPriority[96..127] := 3;
   Std.AlmStruct.BannerPriority[128..159] := 4;
   Std.AlmStruct.BannerPriority[160..191] := 5;
   Std.AlmStruct.BannerPriority[192..1023] := 6;
   Std.AlmStruct.Cause[0..63] := 4;
   Std.AlmStruct.Cause[64..127] := 0;
   Std.AlmStruct.Cause[128..159] := 3;
   Std.AlmStruct.Cause[160..1023] := 4;
   Std.AlmBannerFbk.FirstAlmDetection := FALSE;
   Std.AlmBannerFbk.AlmPriority := 100;
   Std.AlmBannerFbk.AlmCategory := -1;
   Std.AlmBannerFbk.AlmCause := -1;
   Std.AlmBannerFbk.AlmID := -1;
   Std.AlmBannerFbk.GlobalAbsTime := 0;
   Std.SignStruct.Sign[0..31] := 0;
   Std.SignStruct.Category[0..1023] := 0;
   Std.SignStruct.BannerPriority[0..31] := 3;
   Std.SignStruct.BannerPriority[32..63] := 1;
   Std.SignStruct.BannerPriority[64..95] := 2;
   Std.SignStruct.BannerPriority[96..1023] := 0;
   Std.SignBannerFbk.SignPriority := 100;
   Std.SignBannerFbk.SignCategory := -1;
   Std.SignBannerFbk.SignID := -1;
   Std.MaintenanceInput.Clock_1Hz := FALSE;
   Std.MaintenanceInput.CountEnable := FALSE;
   Std.MaintenanceInput.CondToBeActivated := TRUE;
   Std.MaintenanceInput.EventsStrobe := 0;
   Std.LightSiren.Cfg_StaPbt := 65535;
   Std.LightSiren.Cfg_RstPbt := -1;
   Std.LightSiren.Cfg_EnaPbt := 65535;
   Std.LightSiren.Cfg_Siren := 1;
   Std.LightSiren.Cfg_Stack := 1;
   Std.LightSiren.Steady.StaPbtLgh := FALSE;
   Std.LightSiren.Steady.RstPbtLgh := FALSE;
   Std.LightSiren.Steady.EnaPbtLgh := FALSE;
   Std.LightSiren.Steady.Siren := FALSE;
   Std.LightSiren.Steady.YelStkLgh := FALSE;
   Std.LightSiren.Steady.BluStkLgh := FALSE;
   Std.LightSiren.Steady.GrnStkLgh := FALSE;
   Std.LightSiren.Steady.WhtStkLgh := FALSE;
   Std.LightSiren.Steady.Cust1_StaPbtLgh := FALSE;
   Std.LightSiren.Steady.Cust1_RstPbtLgh := FALSE;
   Std.LightSiren.Steady.Cust1_Siren := FALSE;
   Std.LightSiren.Steady.Cust1_RedStkLgh := FALSE;
   Std.LightSiren.Steady.Cust1_OngStkLgh := FALSE;
   Std.LightSiren.Steady.Cust1_GrnStkLgh := FALSE;
   Std.LightSiren.Steady.Cust1_BluStkLgh := FALSE;
   Std.LightSiren.Steady.Cust1_WhtStkLgh := FALSE;
   Std.LightSiren.Frequency1.StaPbtLgh := FALSE;
   Std.LightSiren.Frequency1.RstPbtLgh := FALSE;
   Std.LightSiren.Frequency1.EnaPbtLgh := FALSE;
   Std.LightSiren.Frequency1.Siren := FALSE;
   Std.LightSiren.Frequency1.YelStkLgh := FALSE;
   Std.LightSiren.Frequency1.BluStkLgh := FALSE;
   Std.LightSiren.Frequency1.GrnStkLgh := FALSE;
   Std.LightSiren.Frequency1.WhtStkLgh := FALSE;
   Std.LightSiren.Frequency1.Cust1_StaPbtLgh := FALSE;
   Std.LightSiren.Frequency1.Cust1_RstPbtLgh := FALSE;
   Std.LightSiren.Frequency1.Cust1_Siren := FALSE;
   Std.LightSiren.Frequency1.Cust1_RedStkLgh := FALSE;
   Std.LightSiren.Frequency1.Cust1_OngStkLgh := FALSE;
   Std.LightSiren.Frequency1.Cust1_GrnStkLgh := FALSE;
   Std.LightSiren.Frequency1.Cust1_BluStkLgh := FALSE;
   Std.LightSiren.Frequency1.Cust1_WhtStkLgh := FALSE;
   Std.LightSiren.Frequency2.StaPbtLgh := FALSE;
   Std.LightSiren.Frequency2.RstPbtLgh := FALSE;
   Std.LightSiren.Frequency2.EnaPbtLgh := FALSE;
   Std.LightSiren.Frequency2.Siren := FALSE;
   Std.LightSiren.Frequency2.YelStkLgh := FALSE;
   Std.LightSiren.Frequency2.BluStkLgh := FALSE;
   Std.LightSiren.Frequency2.GrnStkLgh := FALSE;
   Std.LightSiren.Frequency2.WhtStkLgh := FALSE;
   Std.LightSiren.Frequency2.Cust1_StaPbtLgh := FALSE;
   Std.LightSiren.Frequency2.Cust1_RstPbtLgh := FALSE;
   Std.LightSiren.Frequency2.Cust1_Siren := FALSE;
   Std.LightSiren.Frequency2.Cust1_RedStkLgh := FALSE;
   Std.LightSiren.Frequency2.Cust1_OngStkLgh := FALSE;
   Std.LightSiren.Frequency2.Cust1_GrnStkLgh := FALSE;
   Std.LightSiren.Frequency2.Cust1_BluStkLgh := FALSE;
   Std.LightSiren.Frequency2.Cust1_WhtStkLgh := FALSE;
   Std.LightSiren.Frequency3.StaPbtLgh := FALSE;
   Std.LightSiren.Frequency3.RstPbtLgh := FALSE;
   Std.LightSiren.Frequency3.EnaPbtLgh := FALSE;
   Std.LightSiren.Frequency3.Siren := FALSE;
   Std.LightSiren.Frequency3.YelStkLgh := FALSE;
   Std.LightSiren.Frequency3.BluStkLgh := FALSE;
   Std.LightSiren.Frequency3.GrnStkLgh := FALSE;
   Std.LightSiren.Frequency3.WhtStkLgh := FALSE;
   Std.LightSiren.Frequency3.Cust1_StaPbtLgh := FALSE;
   Std.LightSiren.Frequency3.Cust1_RstPbtLgh := FALSE;
   Std.LightSiren.Frequency3.Cust1_Siren := FALSE;
   Std.LightSiren.Frequency3.Cust1_RedStkLgh := FALSE;
   Std.LightSiren.Frequency3.Cust1_OngStkLgh := FALSE;
   Std.LightSiren.Frequency3.Cust1_GrnStkLgh := FALSE;
   Std.LightSiren.Frequency3.Cust1_BluStkLgh := FALSE;
   Std.LightSiren.Frequency3.Cust1_WhtStkLgh := FALSE;
   Std.LightSiren.Frequency4.StaPbtLgh := FALSE;
   Std.LightSiren.Frequency4.RstPbtLgh := FALSE;
   Std.LightSiren.Frequency4.EnaPbtLgh := FALSE;
   Std.LightSiren.Frequency4.Siren := FALSE;
   Std.LightSiren.Frequency4.YelStkLgh := FALSE;
   Std.LightSiren.Frequency4.BluStkLgh := FALSE;
   Std.LightSiren.Frequency4.GrnStkLgh := FALSE;
   Std.LightSiren.Frequency4.WhtStkLgh := FALSE;
   Std.LightSiren.Frequency4.Cust1_StaPbtLgh := FALSE;
   Std.LightSiren.Frequency4.Cust1_RstPbtLgh := FALSE;
   Std.LightSiren.Frequency4.Cust1_Siren := FALSE;
   Std.LightSiren.Frequency4.Cust1_RedStkLgh := FALSE;
   Std.LightSiren.Frequency4.Cust1_OngStkLgh := FALSE;
   Std.LightSiren.Frequency4.Cust1_GrnStkLgh := FALSE;
   Std.LightSiren.Frequency4.Cust1_BluStkLgh := FALSE;
   Std.LightSiren.Frequency4.Cust1_WhtStkLgh := FALSE;
   Std.MachineStateModel.EnableIn := FALSE;
   Std.MachineStateModel.EnableOut := FALSE;
   Std.MachineStateModel.Cmd_Mode := 1;
   Std.MachineStateModel.Cmd_Reset := FALSE;
   Std.MachineStateModel.Cmd_Start := FALSE;
   Std.MachineStateModel.Cmd_Stop := FALSE;
   Std.MachineStateModel.Cmd_Hold := FALSE;
   Std.MachineStateModel.Cmd_UnHold := FALSE;
   Std.MachineStateModel.Cmd_Suspend := FALSE;
   Std.MachineStateModel.Cmd_UnSuspend := FALSE;
   Std.MachineStateModel.Cmd_Abort := FALSE;
   Std.MachineStateModel.Cmd_Clear := FALSE;
   Std.MachineStateModel.Cmd_StateComplete := FALSE;
   Std.MachineStateModel.Cmd_ModeManual := FALSE;
   Std.MachineStateModel.Cmd_ModeProduce := TRUE;
   Std.MachineStateModel.Cfg_RemoteCmdEnable := FALSE;
   Std.MachineStateModel.Inp_RemoteModeCmd := 0;
   Std.MachineStateModel.Inp_RemoteModeCmdChangeRequest := FALSE;
   Std.MachineStateModel.Inp_RemoteStateCmd := 0;
   Std.MachineStateModel.Inp_RemoteStateCmdChangeRequest := FALSE;
   Std.MachineStateModel.StartRequest := FALSE;
   Std.MachineStateModel.ResetRequest := FALSE;
   Std.MachineStateModel.Sts_StateCurrent := 9;
   Std.MachineStateModel.Sts_ModeCurrent := 1;
   Std.MachineStateModel.Sts_DisabledStates := 203776;
   Std.MachineStateModel.Sts_ProductionModeCurrent := TRUE;
   Std.MachineStateModel.Sts_ManualModeCurrent := FALSE;
   Std.MachineStateModel.Sts_ClearingEnabled := TRUE;
   Std.MachineStateModel.Sts_StoppedEnabled := TRUE;
   Std.MachineStateModel.Sts_StartingEnabled := TRUE;
   Std.MachineStateModel.Sts_IdleEnabled := TRUE;
   Std.MachineStateModel.Sts_SuspendedEnabled := TRUE;
   Std.MachineStateModel.Sts_ExecuteEnabled := TRUE;
   Std.MachineStateModel.Sts_StoppingEnabled := TRUE;
   Std.MachineStateModel.Sts_AbortingEnabled := TRUE;
   Std.MachineStateModel.Sts_AbortedEnabled := TRUE;
   Std.MachineStateModel.Sts_HoldingEnabled := FALSE;
   Std.MachineStateModel.Sts_HeldEnabled := FALSE;
   Std.MachineStateModel.Sts_UnHoldingEnabled := FALSE;
   Std.MachineStateModel.Sts_SuspendingEnabled := TRUE;
   Std.MachineStateModel.Sts_UnSuspendingEnabled := TRUE;
   Std.MachineStateModel.Sts_ResettingEnabled := TRUE;
   Std.MachineStateModel.Sts_CompletingEnabled := FALSE;
   Std.MachineStateModel.Sts_CompleteEnabled := FALSE;
   Std.MachineStateModel.Sts_ModeChangeNotAllowed := FALSE;
   Std.MachineStateModel.Sts_Clearing := FALSE;
   Std.MachineStateModel.Sts_Stopped := FALSE;
   Std.MachineStateModel.Sts_Starting := FALSE;
   Std.MachineStateModel.Sts_Idle := FALSE;
   Std.MachineStateModel.Sts_Suspended := FALSE;
   Std.MachineStateModel.Sts_Execute := FALSE;
   Std.MachineStateModel.Sts_Stopping := FALSE;
   Std.MachineStateModel.Sts_Aborting := FALSE;
   Std.MachineStateModel.Sts_Aborted := TRUE;
   Std.MachineStateModel.Sts_Holding := FALSE;
   Std.MachineStateModel.Sts_Held := FALSE;
   Std.MachineStateModel.Sts_UnHolding := FALSE;
   Std.MachineStateModel.Sts_Suspending := FALSE;
   Std.MachineStateModel.Sts_UnSuspending := FALSE;
   Std.MachineStateModel.Sts_Resetting := FALSE;
   Std.MachineStateModel.Sts_Complete := FALSE;
   Std.MachineStateModel.Sts_Completing := FALSE;
   Std.MachineStateModel.Sts_AbortingDone := FALSE;
   Std.MachineStateModel.Sts_ClearingDone := FALSE;
   Std.MachineStateModel.Sts_ResettingDone := FALSE;
   Std.MachineStateModel.Sts_StartingDone := FALSE;
   Std.MachineStateModel.Sts_UnSuspendingDone := FALSE;
   Std.MachineStateModel.Sts_StoppingDone := FALSE;
   Std.MachineStateModel.Sts_SuspendingDone := FALSE;
   Std.MachineStateModel.TON_TimeoutStop.PT := T#0MS;
   Std.MachineStateModel.TON_TimeoutStop.IN := FALSE;
   Std.MachineStateModel.TON_TimeoutAbort.PT := T#0MS;
   Std.MachineStateModel.TON_TimeoutAbort.IN := FALSE;
   Std.MachineStateModel.TON_Start.PT := T#0MS;
   Std.MachineStateModel.TON_Start.IN := FALSE;
   Std.TON_SafetyOn.PT := T#1S;
   Std.TON_SafetyOn.IN := FALSE;
   Std.TOF_SirenEna.PT := T#5S;
   Std.TOF_SirenEna.ET := T#5S;
   Std.TOF_SirenEna.IN := FALSE;
   Param.Gen_Ena_RejectByScale := FALSE;
   Param.Scale_Ena := FALSE;
   Param.Scale_EmptyMould := 1450.0;
   Param.Scale_Setpoint := 1450.0;
   Param.Scale_UpperTolerance := 50.0;
   Param.Scale_LowerTolerance := 50.0;
   Param.Scale_TimePusherOn := 50.0;
   LastHmiDataParam.Gen_Ena_RejectByScale := FALSE;
   LastHmiDataParam.Scale_Ena := FALSE;
   LastHmiDataParam.Scale_EmptyMould := 0.0;
   LastHmiDataParam.Scale_Setpoint := 0.0;
   LastHmiDataParam.Scale_UpperTolerance := 0.0;
   LastHmiDataParam.Scale_LowerTolerance := 0.0;
   LastHmiDataParam.Scale_TimePusherOn := 0.0;
   Alm.ThSwitch."0" := FALSE;   // CW1.Alm.ThSwitch.0
   Alm.ThSwitch."1" := FALSE;   // CW1.Alm.ThSwitch.1
   Alm.ThSwitch."2" := FALSE;   // CW1.Alm.ThSwitch.2
   Alm.ThSwitch."3" := FALSE;   // CW1.Alm.ThSwitch.3
   Alm.ThSwitch."4" := FALSE;   // CW1.Alm.ThSwitch.4
   Alm.ThSwitch."5" := FALSE;   // CW1.Alm.ThSwitch.5
   Alm.ThSwitch."6" := FALSE;   // CW1.Alm.ThSwitch.6
   Alm.ThSwitch."7" := FALSE;   // CW1.Alm.ThSwitch.7
   Alm.ThSwitch."8" := FALSE;   // CW1.Alm.ThSwitch.8
   Alm.ThSwitch."9" := FALSE;   // CW1.Alm.ThSwitch.9
   Alm.ThSwitch."10" := FALSE;   // CW1.Alm.ThSwitch.10
   Alm.ThSwitch."11" := FALSE;   // CW1.Alm.ThSwitch.11
   Alm.ThSwitch."12" := FALSE;   // CW1.Alm.ThSwitch.12
   Alm.ThSwitch."13" := FALSE;   // CW1.Alm.ThSwitch.13
   Alm.ThSwitch."14" := FALSE;   // CW1.Alm.ThSwitch.14
   Alm.ThSwitch."15" := FALSE;   // CW1.Alm.ThSwitch.15
   Alm.ThSwitch."16" := FALSE;   // CW1.Alm.ThSwitch.16
   Alm.ThSwitch."17" := FALSE;   // CW1.Alm.ThSwitch.17
   Alm.ThSwitch."18" := FALSE;   // CW1.Alm.ThSwitch.18
   Alm.ThSwitch."19" := FALSE;   // CW1.Alm.ThSwitch.19
   Alm.ThSwitch."20" := FALSE;   // CW1.Alm.ThSwitch.20
   Alm.ThSwitch."21" := FALSE;   // CW1.Alm.ThSwitch.21
   Alm.ThSwitch."22" := FALSE;   // CW1.Alm.ThSwitch.22
   Alm.ThSwitch."23" := FALSE;   // CW1.Alm.ThSwitch.23
   Alm.ThSwitch."24" := FALSE;   // CW1.Alm.ThSwitch.24
   Alm.ThSwitch."25" := FALSE;   // CW1.Alm.ThSwitch.25
   Alm.ThSwitch."26" := FALSE;   // CW1.Alm.ThSwitch.26
   Alm.ThSwitch."27" := FALSE;   // CW1.Alm.ThSwitch.27
   Alm.ThSwitch."28" := FALSE;   // CW1.Alm.ThSwitch.28
   Alm.ThSwitch."29" := FALSE;   // CW1.Alm.ThSwitch.29
   Alm.ThSwitch."30" := FALSE;   // CW1.Alm.ThSwitch.30
   Alm.ThSwitch."31" := FALSE;   // CW1.Alm.ThSwitch.31
   Alm.SafeComm."0" := FALSE;   // CW1.Alm.SafeComm.0
   Alm.SafeComm."1" := FALSE;   // CW1.Alm.SafeComm.1
   Alm.SafeComm."2" := FALSE;   // CW1.Alm.SafeComm.2
   Alm.SafeComm."3" := FALSE;   // CW1.Alm.SafeComm.3
   Alm.SafeComm."4" := FALSE;   // CW1.Alm.SafeComm.4
   Alm.SafeComm."5" := FALSE;   // CW1.Alm.SafeComm.5
   Alm.SafeComm."6" := FALSE;   // CW1.Alm.SafeComm.6
   Alm.SafeComm."7" := FALSE;   // CW1.Alm.SafeComm.7
   Alm.SafeComm."8" := FALSE;   // CW1.Alm.SafeComm.8
   Alm.SafeComm."9" := FALSE;   // CW1.Alm.SafeComm.9
   Alm.SafeComm."10" := FALSE;   // CW1.Alm.SafeComm.10
   Alm.SafeComm."11" := FALSE;   // CW1.Alm.SafeComm.11
   Alm.SafeComm."12" := FALSE;   // CW1.Alm.SafeComm.12
   Alm.SafeComm."13" := FALSE;   // CW1.Alm.SafeComm.13
   Alm.SafeComm."14" := FALSE;   // CW1.Alm.SafeComm.14
   Alm.SafeComm."15" := FALSE;   // CW1.Alm.SafeComm.15
   Alm.SafeComm."16" := FALSE;   // CW1.Alm.SafeComm.16
   Alm.SafeComm."17" := FALSE;   // CW1.Alm.SafeComm.17
   Alm.SafeComm."18" := FALSE;   // CW1.Alm.SafeComm.18
   Alm.SafeComm."19" := FALSE;   // CW1.Alm.SafeComm.19
   Alm.SafeComm."20" := FALSE;   // CW1.Alm.SafeComm.20
   Alm.SafeComm."21" := FALSE;   // CW1.Alm.SafeComm.21
   Alm.SafeComm."22" := FALSE;   // CW1.Alm.SafeComm.22
   Alm.SafeComm."23" := FALSE;   // CW1.Alm.SafeComm.23
   Alm.SafeComm."24" := FALSE;   // CW1.Alm.SafeComm.24
   Alm.SafeComm."25" := FALSE;   // CW1.Alm.SafeComm.25
   Alm.SafeComm."26" := FALSE;   // CW1.Alm.SafeComm.26
   Alm.SafeComm."27" := FALSE;   // CW1.Alm.SafeComm.27
   Alm.SafeComm."28" := FALSE;   // CW1.Alm.SafeComm.28
   Alm.SafeComm."29" := FALSE;   // CW1.Alm.SafeComm.29
   Alm.SafeComm."30" := FALSE;   // CW1.Alm.SafeComm.30
   Alm.SafeComm."31" := FALSE;   // CW1.Alm.SafeComm.31
   Alm.SafeEmg."0" := FALSE;   // CW1.Alm.SafeEmg.0
   Alm.SafeEmg."1" := FALSE;   // CW1.Alm.SafeEmg.1
   Alm.SafeEmg."2" := FALSE;   // CW1.Alm.SafeEmg.2
   Alm.SafeEmg."3" := FALSE;   // CW1.Alm.SafeEmg.3
   Alm.SafeEmg."4" := FALSE;   // CW1.Alm.SafeEmg.4
   Alm.SafeEmg."5" := FALSE;   // CW1.Alm.SafeEmg.5
   Alm.SafeEmg."6" := FALSE;   // CW1.Alm.SafeEmg.6
   Alm.SafeEmg."7" := FALSE;   // CW1.Alm.SafeEmg.7
   Alm.SafeEmg."8" := FALSE;   // CW1.Alm.SafeEmg.8
   Alm.SafeEmg."9" := FALSE;   // CW1.Alm.SafeEmg.9
   Alm.SafeEmg."10" := FALSE;   // CW1.Alm.SafeEmg.10
   Alm.SafeEmg."11" := FALSE;   // CW1.Alm.SafeEmg.11
   Alm.SafeEmg."12" := FALSE;   // CW1.Alm.SafeEmg.12
   Alm.SafeEmg."13" := FALSE;   // CW1.Alm.SafeEmg.13
   Alm.SafeEmg."14" := FALSE;   // CW1.Alm.SafeEmg.14
   Alm.SafeEmg."15" := FALSE;   // CW1.Alm.SafeEmg.15
   Alm.SafeEmg."16" := FALSE;   // CW1.Alm.SafeEmg.16
   Alm.SafeEmg."17" := FALSE;   // CW1.Alm.SafeEmg.17
   Alm.SafeEmg."18" := FALSE;   // CW1.Alm.SafeEmg.18
   Alm.SafeEmg."19" := FALSE;   // CW1.Alm.SafeEmg.19
   Alm.SafeEmg."20" := FALSE;   // CW1.Alm.SafeEmg.20
   Alm.SafeEmg."21" := FALSE;   // CW1.Alm.SafeEmg.21
   Alm.SafeEmg."22" := FALSE;   // CW1.Alm.SafeEmg.22
   Alm.SafeEmg."23" := FALSE;   // CW1.Alm.SafeEmg.23
   Alm.SafeEmg."24" := FALSE;   // CW1.Alm.SafeEmg.24
   Alm.SafeEmg."25" := FALSE;   // CW1.Alm.SafeEmg.25
   Alm.SafeEmg."26" := FALSE;   // CW1.Alm.SafeEmg.26
   Alm.SafeEmg."27" := FALSE;   // CW1.Alm.SafeEmg.27
   Alm.SafeEmg."28" := FALSE;   // CW1.Alm.SafeEmg.28
   Alm.SafeEmg."29" := FALSE;   // CW1.Alm.SafeEmg.29
   Alm.SafeEmg."30" := FALSE;   // CW1.Alm.SafeEmg.30
   Alm.SafeEmg."31" := FALSE;   // CW1.Alm.SafeEmg.31
   Alm.SafeGuards."0" := FALSE;   // CW1.Alm.SafeGuards.0 > Safe guard 1 open operator side (1AC371BG4)
   Alm.SafeGuards."1" := FALSE;   // CW1.Alm.SafeGuards.1 > Safe guard 2 open not operator side (1AC372BG2)
   Alm.SafeGuards."2" := FALSE;   // CW1.Alm.SafeGuards.2
   Alm.SafeGuards."3" := FALSE;   // CW1.Alm.SafeGuards.3
   Alm.SafeGuards."4" := FALSE;   // CW1.Alm.SafeGuards.4
   Alm.SafeGuards."5" := FALSE;   // CW1.Alm.SafeGuards.5
   Alm.SafeGuards."6" := FALSE;   // CW1.Alm.SafeGuards.6
   Alm.SafeGuards."7" := FALSE;   // CW1.Alm.SafeGuards.7
   Alm.SafeGuards."8" := FALSE;   // CW1.Alm.SafeGuards.8
   Alm.SafeGuards."9" := FALSE;   // CW1.Alm.SafeGuards.9
   Alm.SafeGuards."10" := FALSE;   // CW1.Alm.SafeGuards.10
   Alm.SafeGuards."11" := FALSE;   // CW1.Alm.SafeGuards.11
   Alm.SafeGuards."12" := FALSE;   // CW1.Alm.SafeGuards.12
   Alm.SafeGuards."13" := FALSE;   // CW1.Alm.SafeGuards.13
   Alm.SafeGuards."14" := FALSE;   // CW1.Alm.SafeGuards.14
   Alm.SafeGuards."15" := FALSE;   // CW1.Alm.SafeGuards.15
   Alm.SafeGuards."16" := FALSE;   // CW1.Alm.SafeGuards.16
   Alm.SafeGuards."17" := FALSE;   // CW1.Alm.SafeGuards.17
   Alm.SafeGuards."18" := FALSE;   // CW1.Alm.SafeGuards.18
   Alm.SafeGuards."19" := FALSE;   // CW1.Alm.SafeGuards.19
   Alm.SafeGuards."20" := FALSE;   // CW1.Alm.SafeGuards.20
   Alm.SafeGuards."21" := FALSE;   // CW1.Alm.SafeGuards.21
   Alm.SafeGuards."22" := FALSE;   // CW1.Alm.SafeGuards.22
   Alm.SafeGuards."23" := FALSE;   // CW1.Alm.SafeGuards.23
   Alm.SafeGuards."24" := FALSE;   // CW1.Alm.SafeGuards.24
   Alm.SafeGuards."25" := FALSE;   // CW1.Alm.SafeGuards.25
   Alm.SafeGuards."26" := FALSE;   // CW1.Alm.SafeGuards.26
   Alm.SafeGuards."27" := FALSE;   // CW1.Alm.SafeGuards.27
   Alm.SafeGuards."28" := FALSE;   // CW1.Alm.SafeGuards.28
   Alm.SafeGuards."29" := FALSE;   // CW1.Alm.SafeGuards.29
   Alm.SafeGuards."30" := FALSE;   // CW1.Alm.SafeGuards.30
   Alm.SafeGuards."31" := FALSE;   // CW1.Alm.SafeGuards.31
   Alm.GtaAirGroup."0" := FALSE;   // CW1.Alm.GtaAirGroup.0
   Alm.GtaAirGroup."1" := FALSE;   // CW1.Alm.GtaAirGroup.1
   Alm.GtaAirGroup."2" := FALSE;   // CW1.Alm.GtaAirGroup.2
   Alm.GtaAirGroup."3" := FALSE;   // CW1.Alm.GtaAirGroup.3
   Alm.GtaAirGroup."4" := FALSE;   // CW1.Alm.GtaAirGroup.4
   Alm.GtaAirGroup."5" := FALSE;   // CW1.Alm.GtaAirGroup.5
   Alm.GtaAirGroup."6" := FALSE;   // CW1.Alm.GtaAirGroup.6
   Alm.GtaAirGroup."7" := FALSE;   // CW1.Alm.GtaAirGroup.7
   Alm.GtaAirGroup."8" := FALSE;   // CW1.Alm.GtaAirGroup.8
   Alm.GtaAirGroup."9" := FALSE;   // CW1.Alm.GtaAirGroup.9
   Alm.GtaAirGroup."10" := FALSE;   // CW1.Alm.GtaAirGroup.10
   Alm.GtaAirGroup."11" := FALSE;   // CW1.Alm.GtaAirGroup.11
   Alm.GtaAirGroup."12" := FALSE;   // CW1.Alm.GtaAirGroup.12
   Alm.GtaAirGroup."13" := FALSE;   // CW1.Alm.GtaAirGroup.13
   Alm.GtaAirGroup."14" := FALSE;   // CW1.Alm.GtaAirGroup.14
   Alm.GtaAirGroup."15" := FALSE;   // CW1.Alm.GtaAirGroup.15
   Alm.GtaAirGroup."16" := FALSE;   // CW1.Alm.GtaAirGroup.16
   Alm.GtaAirGroup."17" := FALSE;   // CW1.Alm.GtaAirGroup.17
   Alm.GtaAirGroup."18" := FALSE;   // CW1.Alm.GtaAirGroup.18
   Alm.GtaAirGroup."19" := FALSE;   // CW1.Alm.GtaAirGroup.19
   Alm.GtaAirGroup."20" := FALSE;   // CW1.Alm.GtaAirGroup.20
   Alm.GtaAirGroup."21" := FALSE;   // CW1.Alm.GtaAirGroup.21
   Alm.GtaAirGroup."22" := FALSE;   // CW1.Alm.GtaAirGroup.22
   Alm.GtaAirGroup."23" := FALSE;   // CW1.Alm.GtaAirGroup.23
   Alm.GtaAirGroup."24" := FALSE;   // CW1.Alm.GtaAirGroup.24
   Alm.GtaAirGroup."25" := FALSE;   // CW1.Alm.GtaAirGroup.25
   Alm.GtaAirGroup."26" := FALSE;   // CW1.Alm.GtaAirGroup.26
   Alm.GtaAirGroup."27" := FALSE;   // CW1.Alm.GtaAirGroup.27
   Alm.GtaAirGroup."28" := FALSE;   // CW1.Alm.GtaAirGroup.28
   Alm.GtaAirGroup."29" := FALSE;   // CW1.Alm.GtaAirGroup.29
   Alm.GtaAirGroup."30" := FALSE;   // CW1.Alm.GtaAirGroup.30
   Alm.GtaAirGroup."31" := FALSE;   // CW1.Alm.GtaAirGroup.31
   Alm.Major."0" := FALSE;   // CW1.Alm.Major.0
   Alm.Major."1" := FALSE;   // CW1.Alm.Major.1
   Alm.Major."2" := FALSE;   // CW1.Alm.Major.2
   Alm.Major."3" := FALSE;   // CW1.Alm.Major.3
   Alm.Major."4" := FALSE;   // CW1.Alm.Major.4
   Alm.Major."5" := FALSE;   // CW1.Alm.Major.5
   Alm.Major."6" := FALSE;   // CW1.Alm.Major.6
   Alm.Major."7" := FALSE;   // CW1.Alm.Major.7
   Alm.Major."8" := FALSE;   // CW1.Alm.Major.8
   Alm.Major."9" := FALSE;   // CW1.Alm.Major.9
   Alm.Major."10" := FALSE;   // CW1.Alm.Major.10
   Alm.Major."11" := FALSE;   // CW1.Alm.Major.11
   Alm.Major."12" := FALSE;   // CW1.Alm.Major.12
   Alm.Major."13" := FALSE;   // CW1.Alm.Major.13
   Alm.Major."14" := FALSE;   // CW1.Alm.Major.14
   Alm.Major."15" := FALSE;   // CW1.Alm.Major.15
   Alm.Major."16" := FALSE;   // CW1.Alm.Major.16
   Alm.Major."17" := FALSE;   // CW1.Alm.Major.17
   Alm.Major."18" := FALSE;   // CW1.Alm.Major.18
   Alm.Major."19" := FALSE;   // CW1.Alm.Major.19
   Alm.Major."20" := FALSE;   // CW1.Alm.Major.20
   Alm.Major."21" := FALSE;   // CW1.Alm.Major.21
   Alm.Major."22" := FALSE;   // CW1.Alm.Major.22
   Alm.Major."23" := FALSE;   // CW1.Alm.Major.23
   Alm.Major."24" := FALSE;   // CW1.Alm.Major.24
   Alm.Major."25" := FALSE;   // CW1.Alm.Major.25
   Alm.Major."26" := FALSE;   // CW1.Alm.Major.26
   Alm.Major."27" := FALSE;   // CW1.Alm.Major.27
   Alm.Major."28" := FALSE;   // CW1.Alm.Major.28
   Alm.Major."29" := FALSE;   // CW1.Alm.Major.29
   Alm.Major."30" := FALSE;   // CW1.Alm.Major.30
   Alm.Major."31" := FALSE;   // CW1.Alm.Major.31
   Alm.Minor."0" := FALSE;   // CW1.Alm.Minor.0 > Station in manual mode selected
   Alm.Minor."1" := FALSE;   // CW1.Alm.Minor.1
   Alm.Minor."2" := FALSE;   // CW1.Alm.Minor.2
   Alm.Minor."3" := FALSE;   // CW1.Alm.Minor.3
   Alm.Minor."4" := FALSE;   // CW1.Alm.Minor.4
   Alm.Minor."5" := FALSE;   // CW1.Alm.Minor.5
   Alm.Minor."6" := FALSE;   // CW1.Alm.Minor.6
   Alm.Minor."7" := FALSE;   // CW1.Alm.Minor.7
   Alm.Minor."8" := FALSE;   // CW1.Alm.Minor.8
   Alm.Minor."9" := FALSE;   // CW1.Alm.Minor.9
   Alm.Minor."10" := FALSE;   // CW1.Alm.Minor.10
   Alm.Minor."11" := FALSE;   // CW1.Alm.Minor.11
   Alm.Minor."12" := FALSE;   // CW1.Alm.Minor.12
   Alm.Minor."13" := FALSE;   // CW1.Alm.Minor.13
   Alm.Minor."14" := FALSE;   // CW1.Alm.Minor.14
   Alm.Minor."15" := FALSE;   // CW1.Alm.Minor.15
   Alm.Minor."16" := FALSE;   // CW1.Alm.Minor.16
   Alm.Minor."17" := FALSE;   // CW1.Alm.Minor.17
   Alm.Minor."18" := FALSE;   // CW1.Alm.Minor.18
   Alm.Minor."19" := FALSE;   // CW1.Alm.Minor.19
   Alm.Minor."20" := FALSE;   // CW1.Alm.Minor.20
   Alm.Minor."21" := FALSE;   // CW1.Alm.Minor.21
   Alm.Minor."22" := FALSE;   // CW1.Alm.Minor.22
   Alm.Minor."23" := FALSE;   // CW1.Alm.Minor.23
   Alm.Minor."24" := FALSE;   // CW1.Alm.Minor.24
   Alm.Minor."25" := FALSE;   // CW1.Alm.Minor.25
   Alm.Minor."26" := FALSE;   // CW1.Alm.Minor.26
   Alm.Minor."27" := FALSE;   // CW1.Alm.Minor.27
   Alm.Minor."28" := FALSE;   // CW1.Alm.Minor.28
   Alm.Minor."29" := FALSE;   // CW1.Alm.Minor.29
   Alm.Minor."30" := FALSE;   // CW1.Alm.Minor.30
   Alm.Minor."31" := FALSE;   // CW1.Alm.Minor.31
   Alm.MinorScale."0" := FALSE;   // CW1.Alm.MinorScale.0 > Timeout start condition scale
   Alm.MinorScale."1" := FALSE;   // CW1.Alm.MinorScale.1 > Timeout work scale
   Alm.MinorScale."2" := FALSE;   // CW1.Alm.MinorScale.2 > Thermal switch scale (1ID120QA3)
   Alm.MinorScale."3" := FALSE;   // CW1.Alm.MinorScale.3 > Communication fault scale (1ID120PH7)
   Alm.MinorScale."4" := FALSE;   // CW1.Alm.MinorScale.4 > Scale overload (1ID120PH7)
   Alm.MinorScale."5" := FALSE;   // CW1.Alm.MinorScale.5 > Scale underload (1ID120PH7)
   Alm.MinorScale."6" := FALSE;   // CW1.Alm.MinorScale.6 > Error from scale (1ID120PH7)
   Alm.MinorScale."7" := FALSE;   // CW1.Alm.MinorScale.7 > Timeout tare command (1ID120PH7)
   Alm.MinorScale."8" := FALSE;   // CW1.Alm.MinorScale.8
   Alm.MinorScale."9" := FALSE;   // CW1.Alm.MinorScale.9
   Alm.MinorScale."10" := FALSE;   // CW1.Alm.MinorScale.10 > Scale pusher position not correct (1ID330BG3/4)
   Alm.MinorScale."11" := FALSE;   // CW1.Alm.MinorScale.11
   Alm.MinorScale."12" := FALSE;   // CW1.Alm.MinorScale.12 > Scale in chain obstruction
   Alm.MinorScale."13" := FALSE;   // CW1.Alm.MinorScale.13
   Alm.MinorScale."14" := FALSE;   // CW1.Alm.MinorScale.14
   Alm.MinorScale."15" := FALSE;   // CW1.Alm.MinorScale.15
   Alm.MinorScale."16" := FALSE;   // CW1.Alm.MinorScale.16
   Alm.MinorScale."17" := FALSE;   // CW1.Alm.MinorScale.17
   Alm.MinorScale."18" := FALSE;   // CW1.Alm.MinorScale.18
   Alm.MinorScale."19" := FALSE;   // CW1.Alm.MinorScale.19
   Alm.MinorScale."20" := FALSE;   // CW1.Alm.MinorScale.20
   Alm.MinorScale."21" := FALSE;   // CW1.Alm.MinorScale.21
   Alm.MinorScale."22" := FALSE;   // CW1.Alm.MinorScale.22
   Alm.MinorScale."23" := FALSE;   // CW1.Alm.MinorScale.23
   Alm.MinorScale."24" := FALSE;   // CW1.Alm.MinorScale.24
   Alm.MinorScale."25" := FALSE;   // CW1.Alm.MinorScale.25
   Alm.MinorScale."26" := FALSE;   // CW1.Alm.MinorScale.26
   Alm.MinorScale."27" := FALSE;   // CW1.Alm.MinorScale.27
   Alm.MinorScale."28" := FALSE;   // CW1.Alm.MinorScale.28
   Alm.MinorScale."29" := FALSE;   // CW1.Alm.MinorScale.29
   Alm.MinorScale."30" := FALSE;   // CW1.Alm.MinorScale.30
   Alm.MinorScale."31" := FALSE;   // CW1.Alm.MinorScale.31
   AlmWinCC.ThSwitch[0..1] := 16#0000;
   AlmWinCC.SafeComm[0..1] := 16#0000;
   AlmWinCC.SafeEmg[0..1] := 16#0000;
   AlmWinCC.SafeGuards[0..1] := 16#0000;
   AlmWinCC.GtaAirGroup[0..1] := 16#0000;
   AlmWinCC.Major[0..1] := 16#0000;
   AlmWinCC.Minor[0..1] := 16#0000;
   AlmWinCC.MinorScale[0..1] := 16#0000;
   Sign.General."0" := FALSE;   // CW1.Sign.General.0
   Sign.General."1" := FALSE;   // CW1.Sign.General.1
   Sign.General."2" := FALSE;   // CW1.Sign.General.2
   Sign.General."3" := FALSE;   // CW1.Sign.General.3
   Sign.General."4" := FALSE;   // CW1.Sign.General.4
   Sign.General."5" := FALSE;   // CW1.Sign.General.5
   Sign.General."6" := FALSE;   // CW1.Sign.General.6
   Sign.General."7" := FALSE;   // CW1.Sign.General.7
   Sign.General."8" := FALSE;   // CW1.Sign.General.8
   Sign.General."9" := FALSE;   // CW1.Sign.General.9
   Sign.General."10" := FALSE;   // CW1.Sign.General.10
   Sign.General."11" := FALSE;   // CW1.Sign.General.11
   Sign.General."12" := FALSE;   // CW1.Sign.General.12
   Sign.General."13" := FALSE;   // CW1.Sign.General.13
   Sign.General."14" := FALSE;   // CW1.Sign.General.14
   Sign.General."15" := FALSE;   // CW1.Sign.General.15
   Sign.General."16" := FALSE;   // CW1.Sign.General.16
   Sign.General."17" := FALSE;   // CW1.Sign.General.17
   Sign.General."18" := FALSE;   // CW1.Sign.General.18
   Sign.General."19" := FALSE;   // CW1.Sign.General.19
   Sign.General."20" := FALSE;   // CW1.Sign.General.20
   Sign.General."21" := FALSE;   // CW1.Sign.General.21
   Sign.General."22" := FALSE;   // CW1.Sign.General.22
   Sign.General."23" := FALSE;   // CW1.Sign.General.23
   Sign.General."24" := FALSE;   // CW1.Sign.General.24
   Sign.General."25" := FALSE;   // CW1.Sign.General.25
   Sign.General."26" := FALSE;   // CW1.Sign.General.26
   Sign.General."27" := FALSE;   // CW1.Sign.General.27
   Sign.General."28" := FALSE;   // CW1.Sign.General.28
   Sign.General."29" := FALSE;   // CW1.Sign.General.29
   Sign.General."30" := FALSE;   // CW1.Sign.General.30
   Sign.General."31" := FALSE;   // CW1.Sign.General.31
   Sign.Maintenance_Req."0" := FALSE;   // CW1.Sign.Maintenance_Req.0 > Maintenance 0 request
   Sign.Maintenance_Req."1" := FALSE;   // CW1.Sign.Maintenance_Req.1 > Maintenance 1 request
   Sign.Maintenance_Req."2" := FALSE;   // CW1.Sign.Maintenance_Req.2 > Maintenance 2 request
   Sign.Maintenance_Req."3" := FALSE;   // CW1.Sign.Maintenance_Req.3 > Maintenance 3 request
   Sign.Maintenance_Req."4" := FALSE;   // CW1.Sign.Maintenance_Req.4 > Maintenance 4 request
   Sign.Maintenance_Req."5" := FALSE;   // CW1.Sign.Maintenance_Req.5 > Maintenance 5 request
   Sign.Maintenance_Req."6" := FALSE;   // CW1.Sign.Maintenance_Req.6 > Maintenance 6 request
   Sign.Maintenance_Req."7" := FALSE;   // CW1.Sign.Maintenance_Req.7 > Maintenance 7 request
   Sign.Maintenance_Req."8" := FALSE;   // CW1.Sign.Maintenance_Req.8 > Maintenance 8 request
   Sign.Maintenance_Req."9" := FALSE;   // CW1.Sign.Maintenance_Req.9 > Maintenance 9 request
   Sign.Maintenance_Req."10" := FALSE;   // CW1.Sign.Maintenance_Req.10
   Sign.Maintenance_Req."11" := FALSE;   // CW1.Sign.Maintenance_Req.11
   Sign.Maintenance_Req."12" := FALSE;   // CW1.Sign.Maintenance_Req.12
   Sign.Maintenance_Req."13" := FALSE;   // CW1.Sign.Maintenance_Req.13
   Sign.Maintenance_Req."14" := FALSE;   // CW1.Sign.Maintenance_Req.14
   Sign.Maintenance_Req."15" := FALSE;   // CW1.Sign.Maintenance_Req.15
   Sign.Maintenance_Req."16" := FALSE;   // CW1.Sign.Maintenance_Req.16
   Sign.Maintenance_Req."17" := FALSE;   // CW1.Sign.Maintenance_Req.17
   Sign.Maintenance_Req."18" := FALSE;   // CW1.Sign.Maintenance_Req.18
   Sign.Maintenance_Req."19" := FALSE;   // CW1.Sign.Maintenance_Req.19
   Sign.Maintenance_Req."20" := FALSE;   // CW1.Sign.Maintenance_Req.20
   Sign.Maintenance_Req."21" := FALSE;   // CW1.Sign.Maintenance_Req.21
   Sign.Maintenance_Req."22" := FALSE;   // CW1.Sign.Maintenance_Req.22
   Sign.Maintenance_Req."23" := FALSE;   // CW1.Sign.Maintenance_Req.23
   Sign.Maintenance_Req."24" := FALSE;   // CW1.Sign.Maintenance_Req.24
   Sign.Maintenance_Req."25" := FALSE;   // CW1.Sign.Maintenance_Req.25
   Sign.Maintenance_Req."26" := FALSE;   // CW1.Sign.Maintenance_Req.26
   Sign.Maintenance_Req."27" := FALSE;   // CW1.Sign.Maintenance_Req.27
   Sign.Maintenance_Req."28" := FALSE;   // CW1.Sign.Maintenance_Req.28
   Sign.Maintenance_Req."29" := FALSE;   // CW1.Sign.Maintenance_Req.29
   Sign.Maintenance_Req."30" := FALSE;   // CW1.Sign.Maintenance_Req.30
   Sign.Maintenance_Req."31" := FALSE;   // CW1.Sign.Maintenance_Req.31
   Sign.Maintenance_Activated."0" := FALSE;   // CW1.Sign.Maintenance_Activated.0 > Maintenance 0 activated
   Sign.Maintenance_Activated."1" := FALSE;   // CW1.Sign.Maintenance_Activated.1 > Maintenance 1 activated
   Sign.Maintenance_Activated."2" := FALSE;   // CW1.Sign.Maintenance_Activated.2 > Maintenance 2 activated
   Sign.Maintenance_Activated."3" := FALSE;   // CW1.Sign.Maintenance_Activated.3 > Maintenance 3 activated
   Sign.Maintenance_Activated."4" := FALSE;   // CW1.Sign.Maintenance_Activated.4 > Maintenance 4 activated
   Sign.Maintenance_Activated."5" := FALSE;   // CW1.Sign.Maintenance_Activated.5 > Maintenance 5 activated
   Sign.Maintenance_Activated."6" := FALSE;   // CW1.Sign.Maintenance_Activated.6 > Maintenance 6 activated
   Sign.Maintenance_Activated."7" := FALSE;   // CW1.Sign.Maintenance_Activated.7 > Maintenance 7 activated
   Sign.Maintenance_Activated."8" := FALSE;   // CW1.Sign.Maintenance_Activated.8 > Maintenance 8 activated
   Sign.Maintenance_Activated."9" := FALSE;   // CW1.Sign.Maintenance_Activated.9 > Maintenance 9 activated
   Sign.Maintenance_Activated."10" := FALSE;   // CW1.Sign.Maintenance_Activated.10
   Sign.Maintenance_Activated."11" := FALSE;   // CW1.Sign.Maintenance_Activated.11
   Sign.Maintenance_Activated."12" := FALSE;   // CW1.Sign.Maintenance_Activated.12
   Sign.Maintenance_Activated."13" := FALSE;   // CW1.Sign.Maintenance_Activated.13
   Sign.Maintenance_Activated."14" := FALSE;   // CW1.Sign.Maintenance_Activated.14
   Sign.Maintenance_Activated."15" := FALSE;   // CW1.Sign.Maintenance_Activated.15
   Sign.Maintenance_Activated."16" := FALSE;   // CW1.Sign.Maintenance_Activated.16
   Sign.Maintenance_Activated."17" := FALSE;   // CW1.Sign.Maintenance_Activated.17
   Sign.Maintenance_Activated."18" := FALSE;   // CW1.Sign.Maintenance_Activated.18
   Sign.Maintenance_Activated."19" := FALSE;   // CW1.Sign.Maintenance_Activated.19
   Sign.Maintenance_Activated."20" := FALSE;   // CW1.Sign.Maintenance_Activated.20
   Sign.Maintenance_Activated."21" := FALSE;   // CW1.Sign.Maintenance_Activated.21
   Sign.Maintenance_Activated."22" := FALSE;   // CW1.Sign.Maintenance_Activated.22
   Sign.Maintenance_Activated."23" := FALSE;   // CW1.Sign.Maintenance_Activated.23
   Sign.Maintenance_Activated."24" := FALSE;   // CW1.Sign.Maintenance_Activated.24
   Sign.Maintenance_Activated."25" := FALSE;   // CW1.Sign.Maintenance_Activated.25
   Sign.Maintenance_Activated."26" := FALSE;   // CW1.Sign.Maintenance_Activated.26
   Sign.Maintenance_Activated."27" := FALSE;   // CW1.Sign.Maintenance_Activated.27
   Sign.Maintenance_Activated."28" := FALSE;   // CW1.Sign.Maintenance_Activated.28
   Sign.Maintenance_Activated."29" := FALSE;   // CW1.Sign.Maintenance_Activated.29
   Sign.Maintenance_Activated."30" := FALSE;   // CW1.Sign.Maintenance_Activated.30
   Sign.Maintenance_Activated."31" := FALSE;   // CW1.Sign.Maintenance_Activated.31
   SignWinCC.General[0..1] := 16#0000;
   SignWinCC.Maintenance_Req[0..1] := 16#0000;
   SignWinCC.Maintenance_Activated[0..1] := 16#0000;
   Input.StaPbt := FALSE;
   Input.StoPbt := FALSE;
   Input.RstPbt := FALSE;
   Input.EnaPbt := FALSE;
   Input.Safety.SafeZoneOk := FALSE;
   Input.Safety.Grd_01 := FALSE;
   Input.Safety.Grd_02 := FALSE;
   Output.ModLgh := TRUE;
   ExchangeFromChain.Chain.EnableMove := FALSE;
   ExchangeFromChain.Chain.StrobeWorkReq := FALSE;
   ExchangeFromChain.Chain.StrobeWorkReqMouldBlock := FALSE;
   ExchangeFromChain.Chain.CheckObstruction := TRUE;
   ExchangeFromChain.Chain.MoveInMan := FALSE;
   ExchangeFromChain.Chain.VMasterInPosition := TRUE;
   ExchangeFromChain.Chain.VMasterAtSpeed := FALSE;
   ExchangeFromChain.Chain.Cfg_1Jog_0Move := FALSE;
   ExchangeFromChain.ReqWork.Scale := TRUE;
   ExchangeToChain.Work.Scale := FALSE;
   ExchangeToChain.OutChainObstruction.Scale := TRUE;
   ExchangeToChain.TimeWork.Scale := 0;
   ExchangeToChain.AlmOKImmStopChain := TRUE;
   Scale.ScOk := TRUE;
   Scale.CycleOn := FALSE;
   Scale.Work := FALSE;
   Scale.OkToStop := TRUE;
   Scale.AlmOk := TRUE;
   Scale.OutChainObstruction := TRUE;
   Scale.SingleCycle := FALSE;
   Scale.HighWeight := FALSE;
   Scale.LowWeight := FALSE;
   Scale.Ons_TimeWork := TRUE;
   Scale.Weight := 1497.8;
   Scale.WeightForCheck := 0.0;
   Scale.High_WeightRange := 1500.0;
   Scale.Low_WeightRange := 1400.0;
   Scale.Input.Brk := TRUE;
   Scale.Input.PshOff := TRUE;
   Scale.Input.PshOn := FALSE;
   Scale.Input.Eth.Standstill := TRUE;
   Scale.Input.Eth.Overload := FALSE;
   Scale.Input.Eth.Underload := FALSE;
   Scale.Input.Eth.GenError := FALSE;
   Scale.Input.Eth.ProcessComplete := FALSE;
   Scale.Input.Eth.ProcessOnGoing := FALSE;
   Scale.Input.Eth.ProcessError := FALSE;
   Scale.Input.Eth.NumericValue := 0;
   Scale.Input.Eth.DataFormat := 0;
   Scale.Input.Eth.ParamNum := -1;
   Scale.Input.Eth.ActualWeight := 0.0;
   Scale.Input.Eth.ActualWeightMonitoring := 3991.2;
   Scale.Output.CmdPshOn := FALSE;
   Scale.Output.Eth.Handshake := FALSE;
   Scale.Output.Eth.Write := FALSE;
   Scale.Output.Eth.ResetError := FALSE;
   Scale.Output.Eth.TriggerSignal := 0;
   Scale.Output.Eth.DataFormat := 0;
   Scale.Output.Eth.ParamNum := 0;
   Scale.Output.Eth.NumericValue := 0;
   Scale.Man.Ons_SingleCycle := FALSE;
   Scale.Man.CmdSingleCycle := FALSE;
   Scale.Man.CmdPshOn := FALSE;
   Scale.Man.CmdPshOff := FALSE;
   Scale.Man.EnaPbt := FALSE;
   Scale.Man.RstCmd := TRUE;
   Scale.Man.ScreenNumber := 305_010_301;
   Scale.Man.WithinScreenRange := 0;
   Scale."Step"._00_CycleActivated_CmdPshOn := FALSE;
   Scale."Step"._10_PshOn_CmdPshOff := FALSE;
   Scale."Step"._20_PshOff_CmdRead := FALSE;
   Scale."Step"._30_ReadDone_CmdResetHandShake := FALSE;
   Scale."Step"._40_CycleEnd := FALSE;
   Scale."Step".Ons_StrobeWorkDone := FALSE;
   Scale."Step".StrobeWorkDone := FALSE;
   Scale."Step".ScSeqOk := FALSE;
   Scale."Step".SeqActive := FALSE;
   Scale."Step".TON_WaitingPshOn.PT := T#200MS;
   Scale."Step".TON_WaitingPshOn.IN := FALSE;
   Scale."Step".TON_WaitingPshOff.PT := T#400MS;
   Scale."Step".TON_WaitingPshOff.IN := FALSE;
   Scale.TareStep._00_CycleActivated_CmdTareOn := FALSE;
   Scale.TareStep._10_TareDone_CmdTareOff := FALSE;
   Scale.TareStep._20_CmdSave := FALSE;
   Scale.TareStep._30_SaveDone_CycleEnd := FALSE;
   Scale.TareStep.SeqActive := FALSE;
   Scale.RTO_Work.PT := T#1M;
   Scale.RTO_Work.IN := FALSE;
   Scale.TON_ScOk.PT := T#20S;
   Scale.TON_ScOk.IN := FALSE;
   Scale.TON_TimeoutWork.PT := T#20S;
   Scale.TON_TimeoutWork.IN := FALSE;
   Scale.TON_TimeoutTare.PT := T#20S;
   Scale.TON_TimeoutTare.IN := FALSE;
   Scale.TON_AlmPusher.PT := T#5S;
   Scale.TON_AlmPusher.IN := FALSE;
END_DATA_BLOCK
